FUNCTION_BLOCK ROBOT6TESTFB (* JADE WORKER *)
  (* Standard: 61499-1 *)
  (* Version 1.0, 2014-04-22, Ahmed, Fraunhofer IGD *)
  (* Compiler header: package fb.rt; *)
  (* Compiler Java Sun JDK 1.5.0 *)
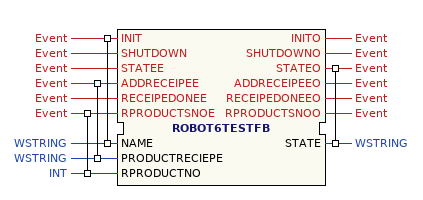
  EVENT_INPUT
    INIT WITH NAME; (* Normal Execution Request *)
    SHUTDOWN;
    STATEE;
    ADDRECEIPEE WITH PRODUCTRECIEPE; (* Normal Execution Request *)
    RECEIPEDONEE;
    RPRODUCTSNOE WITH RPRODUCTNO;
  END_EVENT
  EVENT_OUTPUT
    INITO; (* Execution Confirmation *)
    SHUTDOWNO;
    STATEO WITH STATE;
    ADDRECEIPEEO; (* Execution Confirmation *)
    RECEIPEDONEEO;
    RPRODUCTSNOO;
  END_EVENT
  VAR_INPUT
    NAME : WSTRING;
    PRODUCTRECIEPE : WSTRING;
    RPRODUCTNO : INT;
  END_VAR
  VAR_OUTPUT
    STATE : WSTRING;
  END_VAR
END_FUNCTION_BLOCK
